Xinje XCPPro project, PLC1: XC3-24 (software 3.3L)

PROGRAM Ladder

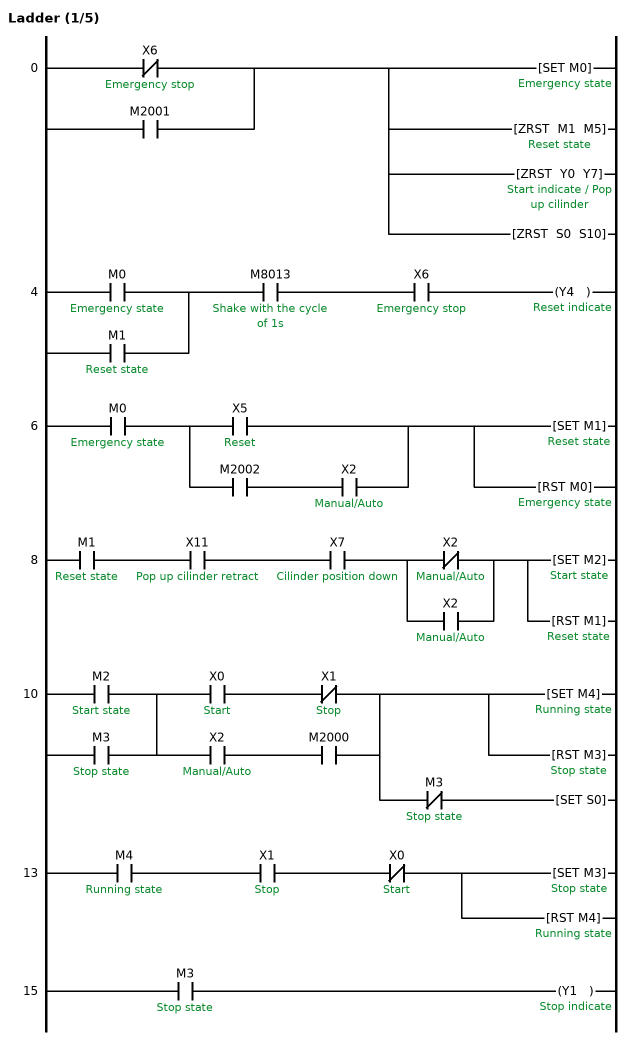
LDI    X6	; Emergency stop
OR     M2001
SET    M0	; Emergency state
ZRST   M1 M5	; Reset state
ZRST   Y0 Y7	; Start indicate / Pop up cilinder
ZRST   S0 S10
LD     M0	; Emergency state
OR     M1	; Reset state
AND    M8013	; Shake with the cycle of 1s
AND    X6	; Emergency stop
OUT    Y4	; Reset indicate
LD     M0	; Emergency state
LD     X5	; Reset
LD     M2002
AND    X2	; Manual/Auto
ORB
ANB
SET    M1	; Reset state
RST    M0	; Emergency state
LD     M1	; Reset state
AND    X11	; Pop up cilinder retract
AND    X7	; Cilinder position down
LDI    X2	; Manual/Auto
OR     X2	; Manual/Auto
ANB
SET    M2	; Start state
RST    M1	; Reset state
LD     M2	; Start state
OR     M3	; Stop state
LD     X0	; Start
ANI    X1	; Stop
LD     X2	; Manual/Auto
AND    M2000
ORB
ANB
SET    M4	; Running state
RST    M3	; Stop state
ANI    M3	; Stop state
SET    S0
LD     M4	; Running state
AND    X1	; Stop
ANI    X0	; Start
SET    M3	; Stop state
RST    M4	; Running state
LD     M3	; Stop state
OUT    Y1	; Stop indicate

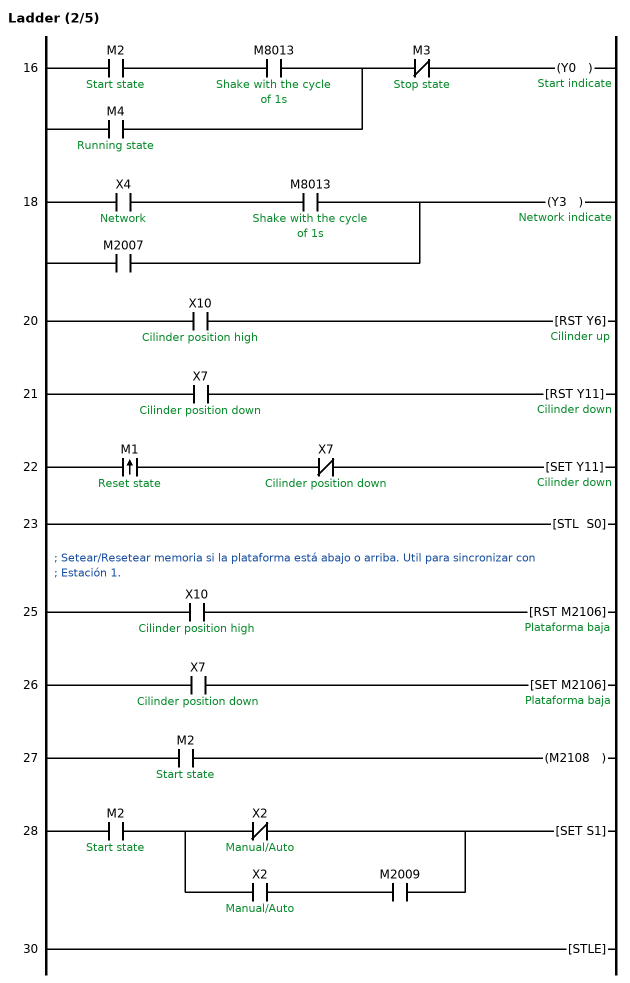
LD     M2	; Start state
AND    M8013	; Shake with the cycle of 1s
OR     M4	; Running state
ANI    M3	; Stop state
OUT    Y0	; Start indicate
LD     X4	; Network
AND    M8013	; Shake with the cycle of 1s
OR     M2007
OUT    Y3	; Network indicate
LD     X10	; Cilinder position high
RST    Y6	; Cilinder up
LD     X7	; Cilinder position down
RST    Y11	; Cilinder down
LDP    M1	; Reset state
ANI    X7	; Cilinder position down
SET    Y11	; Cilinder down
STL    S0
;  Setear/Resetear memoria si la plataforma está abajo o arriba. Util para sincronizar con Estación 1.
LD     X10	; Cilinder position high
RST    M2106	; Plataforma baja
LD     X7	; Cilinder position down
SET    M2106	; Plataforma baja
LD     M2	; Start state
OUT    M2108
LD     M2	; Start state
LDI    X2	; Manual/Auto
LD     X2	; Manual/Auto
AND    M2009
ORB
ANB
SET    S1
STLE

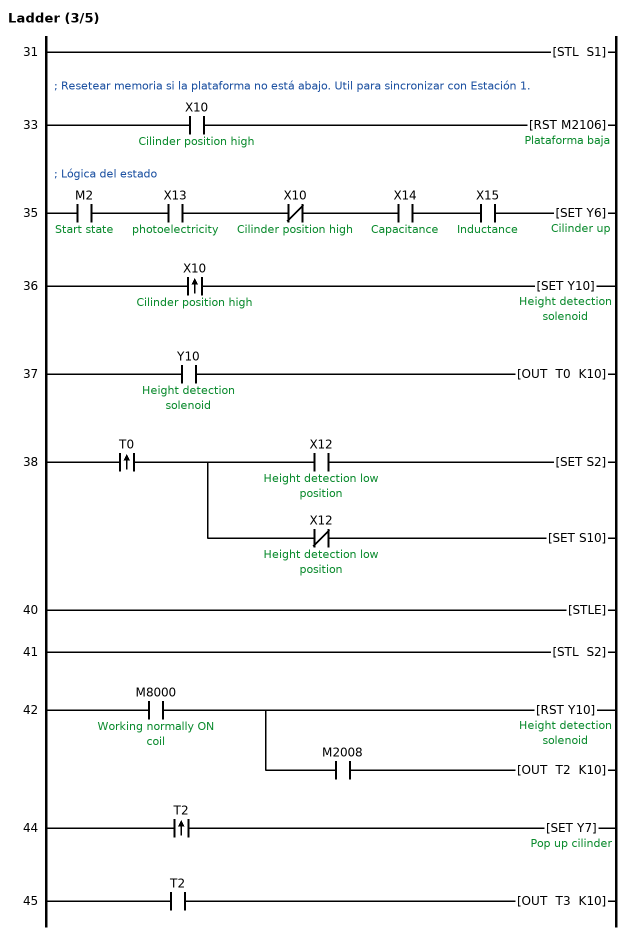
STL    S1
;  Resetear memoria si la plataforma no está abajo. Util para sincronizar con Estación 1.
LD     X10	; Cilinder position high
RST    M2106	; Plataforma baja
;  Lógica del estado
LD     M2	; Start state
AND    X13	; photoelectricity
ANI    X10	; Cilinder position high
AND    X14	; Capacitance
AND    X15	; Inductance
SET    Y6	; Cilinder up
LDP    X10	; Cilinder position high
SET    Y10	; Height detection solenoid
LD     Y10	; Height detection solenoid
OUT    T0 K10
LDP    T0
MPS
AND    X12	; Height detection low position
SET    S2
MPP
ANI    X12	; Height detection low position
SET    S10
STLE
STL    S2
LD     M8000	; Working normally ON coil
RST    Y10	; Height detection solenoid
AND    M2008
OUT    T2 K10
LDP    T2
SET    Y7	; Pop up cilinder
LD     T2
OUT    T3 K10

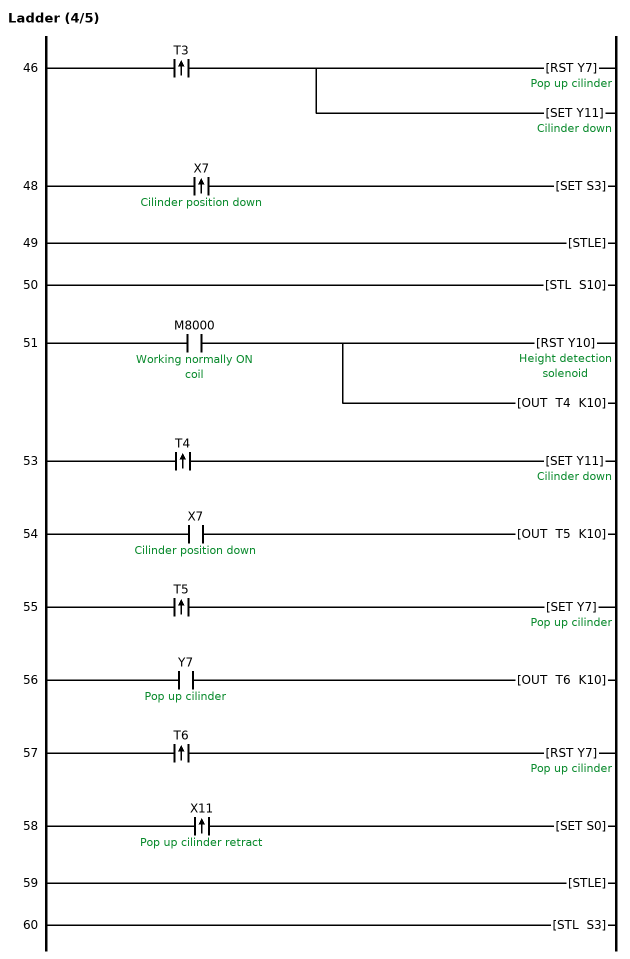
LDP    T3
RST    Y7	; Pop up cilinder
SET    Y11	; Cilinder down
LDP    X7	; Cilinder position down
SET    S3
STLE
STL    S10
LD     M8000	; Working normally ON coil
RST    Y10	; Height detection solenoid
OUT    T4 K10
LDP    T4
SET    Y11	; Cilinder down
LD     X7	; Cilinder position down
OUT    T5 K10
LDP    T5
SET    Y7	; Pop up cilinder
LD     Y7	; Pop up cilinder
OUT    T6 K10
LDP    T6
RST    Y7	; Pop up cilinder
LDP    X11	; Pop up cilinder retract
SET    S0
STLE
STL    S3

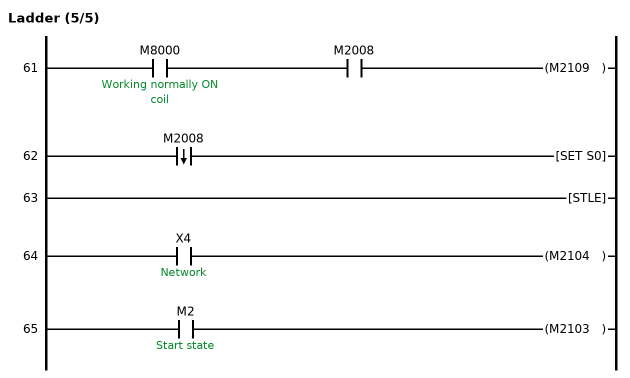
LD     M8000	; Working normally ON coil
AND    M2008
OUT    M2109
LDF    M2008
SET    S0
STLE
LD     X4	; Network
OUT    M2104
LD     M2	; Start state
OUT    M2103

COMMENTS (devices not used above)
X3	Height detection high position
Y5	Alarm indicate